// TIA Portal V17 export
// export: Created 2025-06-26T06:49:32.404206Z, ExportSetting WithDefaults, DisplayName Totally Integrated Automation Portal, DisplayVersion V17 Update 8, DisplayName TIA Portal Openness, DisplayVersion V17 Update 8, DisplayName TIA Portal Version Control Interface, DisplayVersion V17, DisplayName STEP 7 Professional, DisplayVersion V17 Update 8, DisplayName STEP 7 Safety, DisplayVersion V17 Update 6, DisplayName WinCC Advanced, DisplayVersion V17 Update 8
TYPE "StaticSetting-STRUCT"
// stored: IsFailsafeCompliant false
   STRUCT
      AdditionalSuperHeatOnColdStart { ExternalWritable := 'False'} : Real;
      Limits { ExternalWritable := 'False'} : Struct
         T_Ambient_Max { ExternalWritable := 'False'} : Real := 40.0;
         T_Cabinet_Max { ExternalWritable := 'False'} : Real := 45.0;
      END_STRUCT;
   END_STRUCT;
END_TYPE
